// TIA Portal V20 export
TYPE "Log_Data_Byte_Decimal"
// stored: Namespace ProductionLine
   STRUCT
      DataType : Int;
      Representation : Int;
      RepreLength : Int;
      Reserve : Int;
      Data : Int;
   END_STRUCT;
END_TYPE
